FUNCTION_BLOCK T_TcpSend
VAR
	sender : FB_SocketSend;
	_socket : REFERENCE TO T_HSOCKET;	// TCP-IP socket
	_log : T_NamedBase;
	_message : T_MAXSTRING;				// Message to send
END_VAR

METHOD PUBLIC CyclicLogic
IF NOT __ISVALIDREF(_socket) THEN
  RETURN;
END_IF

sender(
	sSrvNetId:= , 
	hSocket:= _socket, 
	cbLen:= TO_UDINT(LEN(_message)), 
	pSrc:= ADR(_message), 
	bExecute:= , 
	tTimeout:= TimeOut, 
	bBusy=> , 
	bError=> , 
	nErrId=> );

IF NOT sender.bBusy THEN
  sender.bExecute := FALSE;
END_IF

IF sender.bError THEN
	_log.LogError('Send Error');
END_IF
END_METHOD

PROPERTY ErrID : UDINT
GET
ErrID := sender.nErrId;
END_GET
END_PROPERTY

PROPERTY INTERNAL HasSocket : BOOL
GET
HasSocket := __ISVALIDREF(_socket);
END_GET
END_PROPERTY

PROPERTY PUBLIC IsBusy : BOOL
GET
IsBusy := sender.bBusy;
END_GET
END_PROPERTY

PROPERTY PUBLIC IsError : BOOL
GET
IsError := sender.bError;
END_GET
END_PROPERTY

METHOD PUBLIC Send : BOOL;
VAR_INPUT
  message : T_MAXSTRING; 
END_VAR
IF NOT HasSocket THEN
  _log.LogError('Cannot Send as NOT HasSocket');
  RETURN;

END_IF

_message := message;
sender.bExecute := TRUE;
Send := TRUE;
END_METHOD

METHOD INTERNAL SetSocket : BOOL
VAR_IN_OUT
  socket : T_HSOCKET;
END_VAR
_socket REF= socket;
_log.LogDebug('SetSocket := TRUE');
SetSocket := TRUE;
END_METHOD

END_FUNCTION_BLOCK

(* stored: Version 1.1.0.1
   POU T_TcpSend: Id {77962015-4eaf-4782-8a73-a6c6e369ba80}, SpecialFunc None
   Folder Methods: Id {b0a6419d-7403-4f4e-94c3-f59fe72f21df}
   Folder Properties: Id {ac29a6d0-5ee4-4e08-a3d9-3eb656b8c981}
   Method CyclicLogic: Id {ac3c3310-df7f-406d-be73-c9b4ce7d7a04}
   Property ErrID: Id {c47b9c96-b7d6-4cda-b920-e7266e016f6f}
   Get Get: Id {ca95efa7-a56b-46f4-95ac-c76f408774da}
   Property HasSocket: Id {cd0135b7-1b06-48c1-90d9-bb4580a65c7b}
   Get Get: Id {cf6d40c3-6a1f-41f1-86e2-b12b24c4c714}
   Property IsBusy: Id {06cdc633-c504-4117-a331-b914d1da7da6}
   Get Get: Id {f731220c-a269-4699-b614-776b87a392ca}
   Property IsError: Id {b125c8c6-3bc1-469a-a40c-c9bf25309665}
   Get Get: Id {b4a2bf1b-176b-4560-89d7-b336e18f7bc4}
   Method Send: Id {16968662-be37-487b-aeee-a7f97a741529}
   Method SetSocket: Id {9a88923a-f0d1-4ccd-983a-26d9df27af99} *)
